// LS Electric XG5000 project: PLC_2차 프로젝트
// PLC PLC_인버터제어
// module base 0 slot 0: 입출력 모듈:XBC-DR32H (DC 24V 입력, 릴레이 출력 32점)

PROGRAM 01_Conveyor_Belt (task: 스캔 프로그램)

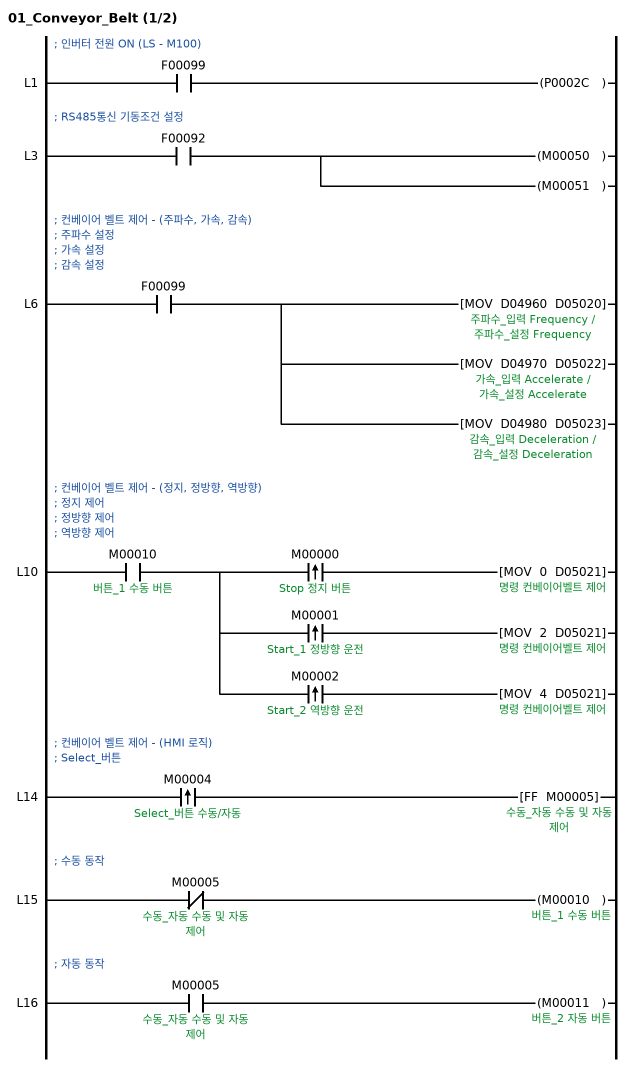
// 인버터 전원 ON (LS - M100)
; L1
LOAD      F00099
OUT       P0002C
// RS485통신 기동조건 설정
; L3
LOAD      F00092
OUT       M00050
OUT       M00051
// 컨베이어 벨트 제어 - (주파수, 가속, 감속)
; L6
LOAD      F00099
MOV       D04960 D05020	// 주파수_입력 Frequency / 주파수_설정 Frequency
MOV       D04970 D05022	// 가속_입력 Accelerate / 가속_설정 Accelerate
MOV       D04980 D05023	// 감속_입력 Deceleration / 감속_설정 Deceleration
// output comment: 주파수 설정
// output comment: 가속 설정
// output comment: 감속 설정
// 컨베이어 벨트 제어 - (정지, 정방향, 역방향)
; L10
LOAD      M00010	// 버튼_1 수동 버튼
MPUSH
ANDP      M00000	// Stop 정지 버튼
MOV       0 D05021	// 명령 컨베이어벨트 제어
MLOAD
ANDP      M00001	// Start_1 정방향 운전
MOV       2 D05021	// 명령 컨베이어벨트 제어
MPOP
ANDP      M00002	// Start_2 역방향 운전
MOV       4 D05021	// 명령 컨베이어벨트 제어
// output comment: 정지 제어
// output comment: 정방향 제어
// output comment: 역방향 제어
// 컨베이어 벨트 제어 - (HMI 로직)
; L14
LOADP     M00004	// Select_버튼 수동/자동
FF        M00005	// 수동_자동 수동 및 자동 제어
// output comment: Select_버튼
; L15
LOAD NOT  M00005	// 수동_자동 수동 및 자동 제어
OUT       M00010	// 버튼_1 수동 버튼
// output comment: 수동 동작
; L16
LOAD      M00005	// 수동_자동 수동 및 자동 제어
OUT       M00011	// 버튼_2 자동 버튼
// output comment: 자동 동작

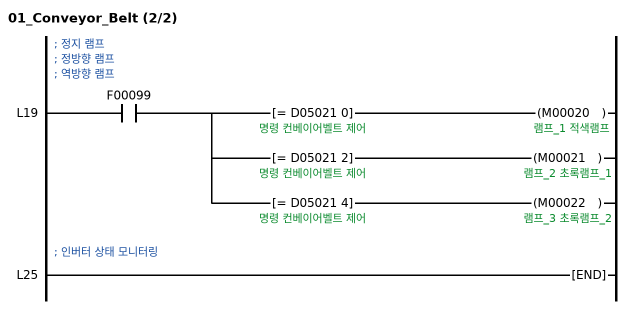
; L19
LOAD      F00099
MPUSH
AND=      D05021 0	// 명령 컨베이어벨트 제어
OUT       M00020	// 램프_1 적색램프
MLOAD
AND=      D05021 2	// 명령 컨베이어벨트 제어
OUT       M00021	// 램프_2 초록램프_1
MPOP
AND=      D05021 4	// 명령 컨베이어벨트 제어
OUT       M00022	// 램프_3 초록램프_2
// output comment: 정지 램프
// output comment: 정방향 램프
// output comment: 역방향 램프
// 인버터 상태 모니터링
; L25
END

PROGRAM 02_Sensor (task: 스캔 프로그램)

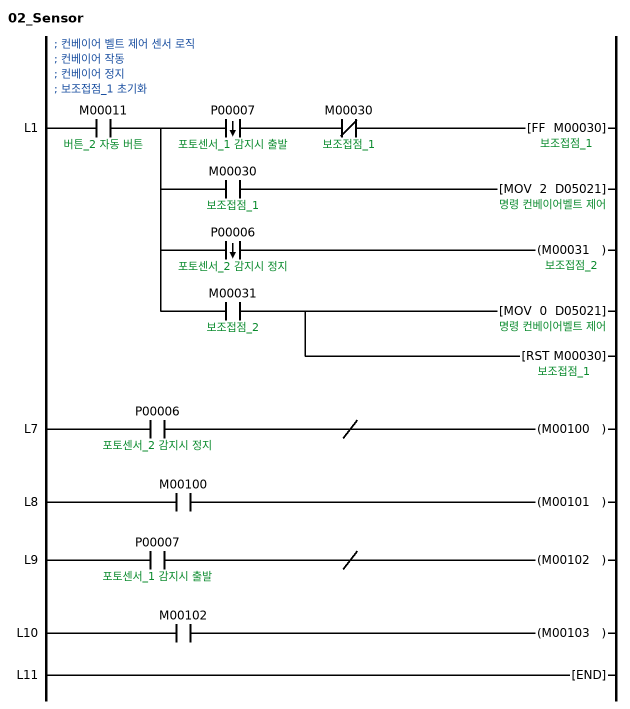
// 컨베이어 벨트 제어 센서 로직
; L1
LOAD      M00011	// 버튼_2 자동 버튼
MPUSH
ANDN      P00007	// 포토센서_1 감지시 출발
AND NOT   M00030	// 보조접점_1
FF        M00030	// 보조접점_1
MLOAD
AND       M00030	// 보조접점_1
MOV       2 D05021	// 명령 컨베이어벨트 제어
MLOAD
ANDN      P00006	// 포토센서_2 감지시 정지
OUT       M00031	// 보조접점_2
MPOP
AND       M00031	// 보조접점_2
MOV       0 D05021	// 명령 컨베이어벨트 제어
RST       M00030	// 보조접점_1
// output comment: 컨베이어 작동
// output comment: 컨베이어 정지
// output comment: 보조접점_1 초기화
; L7
LOAD      P00006	// 포토센서_2 감지시 정지
NOT
OUT       M00100
; L8
LOAD      M00100
OUT       M00101
; L9
LOAD      P00007	// 포토센서_1 감지시 출발
NOT
OUT       M00102
; L10
LOAD      M00102
OUT       M00103
; L11
END

VARIABLES AND COMMENTS (devices not used above)
M00006	BIT	자동 // 자동 제어